(* IEC 61131-3 sources: com.logicals.lc3.webinar/usRTS_RPMControl_iSOC/src_FB_LIB_SAFE/Convert/DINT, 4 files *)

(* ---- wDINT_TO_LINT.iecst ---- *)
NAMESPACE logicals.web.standard
NAMESPACE convert

/*
 * Function block wrapper for IEC 61131-3 TO_LINT<br>
 * IN =  input value (DINT)<br>
 * OUT = IN (LINT)<br>
 */
FUNCTION_BLOCK wDINT_TO_LINT
	{ vNameAlignment:="center"; altName:="DINT_TO_LINT"; bgColor:="LightPink"; width:=140; hideIONames; }
	VAR_INPUT
		IN : DINT;
	END_VAR
	VAR_OUTPUT
		OUT: LINT;
	END_VAR

	OUT := TO_LINT(IN:=IN, ENO=>ENO);
END_FUNCTION_BLOCK

END_NAMESPACE
END_NAMESPACE

(* ---- wTRUNC_DINT_TO_INT.iecst ---- *)
NAMESPACE logicals.web.standard
NAMESPACE convert

/*
 * Function block wrapper for IEC 61131-3 TO_INT<br>
 * IN =  input value (DINT)<br>
 * OUT = IN (INT)<br>
 */
FUNCTION_BLOCK wTRUNC_DINT_TO_INT
	{ vNameAlignment:="center"; altName:="TRUNC_DINT_TO_INT"; bgColor:="LightPink"; width:=180; hideIONames; }
	VAR_INPUT
		IN : DINT;
	END_VAR
	VAR_OUTPUT
		OUT: INT;
	END_VAR

	OUT := TO_INT(IN:=IN, ENO=>ENO);
END_FUNCTION_BLOCK

END_NAMESPACE
END_NAMESPACE

(* ---- wTRUNC_DINT_TO_SINT.iecst ---- *)
NAMESPACE logicals.web.standard
NAMESPACE convert

/*
 * Function block wrapper for IEC 61131-3 TO_SINT<br>
 * IN =  input value (DINT)<br>
 * OUT = IN (SINT)<br>
 */
FUNCTION_BLOCK wTRUNC_DINT_TO_SINT
	{ vNameAlignment:="center"; altName:="TRUNC_DINT_TO_SINT"; bgColor:="LightPink"; width:=180; hideIONames; }
	VAR_INPUT
		IN : DINT;
	END_VAR
	VAR_OUTPUT
		OUT: SINT;
	END_VAR

	OUT := TO_SINT(IN:=IN, ENO=>ENO);
END_FUNCTION_BLOCK

END_NAMESPACE
END_NAMESPACE

(* ---- wTRUNC_DINT_TO_UDINT.iecst ---- *)
NAMESPACE logicals.web.standard
NAMESPACE convert

/*
 * Function block wrapper for IEC 61131-3 TO_UDINT<br>
 * IN =  input value (DINT)<br>
 * OUT = IN (UDINT)<br>
 */
FUNCTION_BLOCK wTRUNC_DINT_TO_UDINT
	{ vNameAlignment:="center"; altName:="TRUNC_DINT_TO_UDINT"; bgColor:="Plum"; width:=180; hideIONames; }
	VAR_INPUT
		IN : DINT;
	END_VAR
	VAR_OUTPUT
		OUT: UDINT;
	END_VAR

	OUT := TO_UDINT(IN:=IN, ENO=>ENO);
END_FUNCTION_BLOCK

END_NAMESPACE
END_NAMESPACE
